PROGRAM PositionVerAxis
VAR
END_VAR

VAVL.axis.ReadStatus();

VAVL.axisPower(
	Axis:= VAVL.axis,
	Enable:= VAVL.enable,
	Enable_Positive:= VAVL.enable,
	Enable_Negative:= VAVL.enable,
	Override:= VAVL.override,
	BufferMode:= ,
	Options:= ,
	Status=> VAVL.running,
	Busy=> ,
	Active=> ,
	Error=> ,
	ErrorID=> VAVL.currentErrorPower
);

VAVL.axisMoveAbsolute(
	Axis:= VAVL.axis,
	Execute:= VAVL.enableMove,
	Position:= VAVL.targetPosition,
	Velocity:= VAVL.targetVelocity,
	Acceleration:= ,
	Deceleration:= ,
	Jerk:= ,
	BufferMode:= ,
	Options:= ,
	Done=> VAVL.done,
	Busy=> VAVL.busy,
	Active=> ,
	CommandAborted=> ,
	Error=> ,
	ErrorID=> VAVL.currentErrorCommand 
);

IF VAVL.busy THEN
	VAVL.axisReadActualPosition(Axis := VAVL.axis, Enable := TRUE, Valid=>, Busy=>, Error=>, ErrorID=>, Position=> VAVL.actualPosition);
END_IF
VAVL.actualPositionInt := LREAL_TO_INT(VAVL.actualPosition);

VAVL.axisErrorReset(Axis := VAVL.axis, Execute := VAVL.resetError, Done =>, Error =>, ErrorID => VAVL.currentError);

END_PROGRAM

(* stored: Version 1.1.0.1, ProductVersion 3.1.4024.6
   POU PositionVerAxis: Id {1b6ad884-2529-406e-ba25-f2207e3320ae}, SpecialFunc None *)
